Universal Robots PolyScope program: PSA_Tatiana.urp

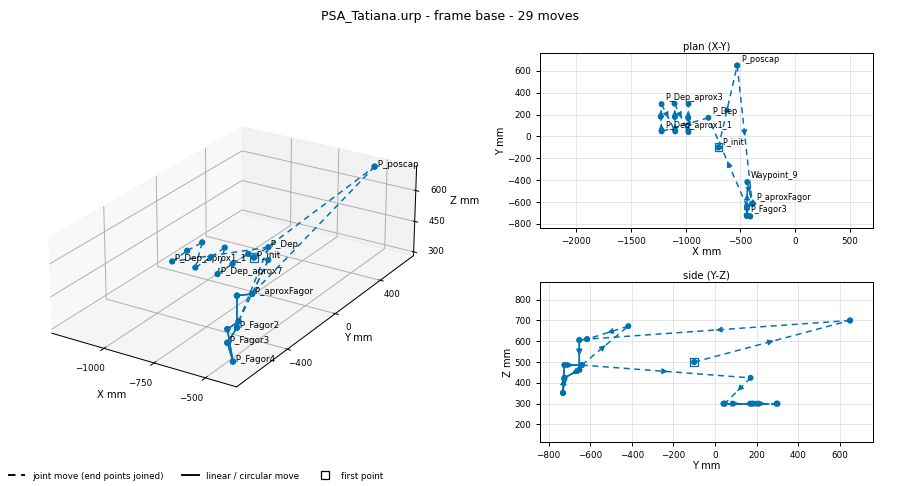
[picture p0: tool path of PSA_Tatiana.urp in frame base, 29 of 35 moves have a stored position in this frame; points joined in program order, loops and branches not executed]
Program PSA_Tatiana (installation=fbarreto directory=/programs/usbdisk createdIn=3.1.17195.0 lastSavedIn=3.15.3.106223 robotSerialNumber=2016302743)
Calibrated DH parameters: a=[0.000062, -0.599238, -0.569293, -0.000071, 0.00007, 0]; d=[0.127903, 43.80973, -52.244011, 8.598345, 0.115597, 0.092059]; alpha=[1.570295, -0.002885, -0.005578, 1.570526, -1.570968, 0]; deltaTheta=[0, -0.207803, 0.290321, -0.082351, -0.000076, 0.000026]
BeforeStart
  Set DigitalOutput pin=digital_out[1]; digitalValue=0
  RecolherPeca := False
  Set DigitalOutput pin=digital_out[2]; digitalValue=0
  RetirarPeca := False
  open := socket_open("192.168.114.51",5024)
  Loop While (checkContinuously=false) expression=open≟ False
    open := socket_open("192.168.114.51",5024)
  targetPos := p[0,0,0,0,0,0]
  '# Configuracao variaveis'
  var_from := p[0,0,0.05,0,0,0]
  var_from := p[0,0,-0.05,0,0,0]
  var_from := p[0.1,0,0,0,0,0]
  var_from := p[-0.1,0,0,0,0,0]
  P_dep_des := p[0,0,150/1000,0,0,0]
  P_dep_sub := p[0,0,-150/1000,0,0,0]
Robot Program (runOnlyOnce=false)
  '# Ligar Camara'
  Loop While (checkContinuously=false) expression=open≟ False
    open := socket_open("192.168.114.51",5024)
  Set DigitalOutput pin=digital_out[1]; digitalValue=1
  MoveJ speed 60 deg/s, acceleration 80 deg/s^2 (useActiveTCP=true)
    Waypoint P_init: TCP in base x=-700 y=-100 z=500 mm, rx=3.14 ry=0 rz=0 rad; joints [-5.413, -88.076, 103.177, -105.112, -90.206, -275.345] deg
    Loop While (checkContinuously=false) expression=RecolherPeca≟ False
      RecolherPeca := read_input_boolean_register(0)
    Waypoint P_poscap: TCP in base x=-528.533 y=649.105 z=699.93 mm, rx=2.2433 ry=-2.1967 rz=0 rad; joints [-62.276, -76.967, 70.287, -83.309, -90.248, -243.289] deg
  receiveFromServ := [0,0,0,0,0,0,0]
  SuppressedNode
    Wait Sleep waitTime=2
  receiveFromServ := socket_read_ascii_float(6)
  Loop While (checkContinuously=false) expression=receiveFromServ[0]≠6
    Wait Sleep waitTime=2
    sendToServer := "10@"
    Script: socket_send_string(sendToServer)
    receiveFromServ := socket_read_ascii_float(6)
  Folder GetCameraData Folder
    '# Here we should read the data from the camera'
    Ry := receiveFromServ[4]
    x_cam := receiveFromServ[2]
    y_cam := receiveFromServ[3]
    NewX := receiveFromServ[5]
    NewY := receiveFromServ[6]
  Folder Calculate Folder
    '# Convert mm to m and deg to rad'
    SuppressedNode
      Script file /programs/PSA_Tati_Pos.script
        | x=x_cam-x_cam*cos(Ry)
    target1 := p[x_cam/1000,y_cam/1000,0,0,0,0]
    target2 := p[0,0,0,0,0,Ry]
    target3 := p[NewX/1000,NewY/1000,0,0,0,0]
    target4 := p[0,0,285/1000,0,0,0]
  Folder MoveToCamPose
    MoveL speed 250 mm/s, acceleration 1200 mm/s^2 (useActiveTCP=false) tcp=TCP; feature=Joint_6_name
      Waypoint Waypoint (Variable): variable=target1
      Wait Sleep waitTime=0.5
      Waypoint Waypoint (Variable): variable=target2
      Wait Sleep waitTime=0.5
      Waypoint Waypoint (Variable): variable=target3
      Wait Sleep waitTime=0.5
      Waypoint Waypoint (Variable): variable=target4
      Set DigitalOutput pin=Ar; digitalValue=1
      Wait Sleep waitTime=2
      Waypoint P_poscap: motionParameters(blendRadius=0.05); TCP in base x=-528.533 y=649.105 z=699.93 mm, rx=2.2433 ry=-2.1967 rz=0 rad; joints [-62.276, -76.967, 70.287, -83.309, -90.248, -243.289] deg; pose in feature x=0 y=0 z=0 mm, rx=0 ry=0 rz=0 rad
  'Registo para PLC'
  Set DigitalOutput pin=digital_out[2]; digitalValue=1
  RecolherPeca := False
  Wait Sleep waitTime=0.1
  Set DigitalOutput pin=digital_out[2]; digitalValue=0
  'Movimentos para Fagor'
  MoveJ speed 60 deg/s, acceleration 80 deg/s^2 (useActiveTCP=true)
    SuppressedNode
      Waypoint P_init: TCP in base x=-700 y=-100 z=500 mm, rx=3.14 ry=0 rz=0 rad; joints [-5.413, -88.076, 103.177, -105.112, -90.206, -275.345] deg
    Waypoint P_aproxFagor: motionParameters(blendRadius=0.01); TCP in base x=-390.993 y=-615.089 z=610.275 mm, rx=2.1894 ry=-2.2258 rz=-0.0638 rad; joints [44.727, -87.76, 91.848, -95.173, -92.658, -134.226] deg
  MoveL speed 250 mm/s, acceleration 1200 mm/s^2 (useActiveTCP=true) feature=Base
    Waypoint P_Fagor1: motionParameters(blendRadius=0.05); TCP in base x=-439.397 y=-652.65 z=605.5 mm, rx=2.1896 ry=-2.2257 rz=-0.0637 rad; joints [44.175, -82.193, 86.245, -95.154, -92.662, -134.786] deg
    Waypoint P_Fagor2: motionParameters(blendRadius=0.05); TCP in base x=-439.462 y=-652.642 z=462.779 mm, rx=2.1897 ry=-2.2257 rz=-0.0637 rad; joints [44.183, -79.624, 97.856, -109.336, -92.647, -134.857] deg
    Waypoint P_Fagor3: motionParameters(blendRadius=0.029); TCP in base x=-440.419 y=-723.918 z=424.353 mm, rx=2.1893 ry=-2.2258 rz=-0.0638 rad; joints [47.686, -72.933, 93.423, -111.459, -92.725, -131.351] deg
    Waypoint P_Fagor4: TCP in base x=-409.469 y=-731.178 z=351.347 mm, rx=2.1897 ry=-2.2256 rz=-0.0643 rad; joints [49.639, -70.944, 98.714, -118.649, -92.761, -129.448] deg
    Set DigitalOutput pin=Ar; digitalValue=0
    Waypoint P_Fagor5: TCP in base x=-440.242 y=-724.015 z=485.586 mm, rx=2.1897 ry=-2.2257 rz=-0.0637 rad; joints [47.695, -74.653, 89.238, -105.541, -92.728, -131.322] deg
    Waypoint P_Fagor6: TCP in base x=-439.303 y=-640.298 z=485.545 mm, rx=2.1898 ry=-2.2259 rz=-0.0638 rad; joints [43.522, -81.208, 97.348, -107.258, -92.636, -135.506] deg
  'Registo para PLC'
  Set DigitalOutput pin=digital_out[3]; digitalValue=1
  Wait Sleep waitTime=0.1
  Set DigitalOutput pin=digital_out[3]; digitalValue=0
  'Esperar Maquinacao'
  MoveJ speed 60 deg/s, acceleration 80 deg/s^2 (useActiveTCP=true)
    Waypoint Waypoint_9: TCP in base x=-436.536 y=-416.989 z=672.545 mm, rx=2.1898 ry=-2.2258 rz=-0.0637 rad; joints [28.076, -100.049, 97.106, -88.753, -92.228, -150.869] deg
  Loop While (checkContinuously=false) expression=RetirarPeca≟ False
    RetirarPeca := read_input_boolean_register(2)
  SuppressedNode
    Wait Sleep waitTime=5
  MoveJ speed 60 deg/s, acceleration 80 deg/s^2 (useActiveTCP=true)
    SuppressedNode
      Waypoint P_init: TCP in base x=-700 y=-100 z=500 mm, rx=3.14 ry=0 rz=0 rad; joints [-5.413, -88.076, 103.177, -105.112, -90.206, -275.345] deg
    Waypoint P_aproxFagor: TCP in base x=-390.993 y=-615.089 z=610.275 mm, rx=2.1894 ry=-2.2258 rz=-0.0638 rad; joints [44.727, -87.76, 91.848, -95.173, -92.658, -134.226] deg
  MoveL speed 250 mm/s, acceleration 1200 mm/s^2 (useActiveTCP=true) feature=Base
    Waypoint P_Fagor1_1: motionParameters(blendRadius=0.05); TCP in base x=-439.397 y=-652.65 z=605.5 mm, rx=2.1896 ry=-2.2257 rz=-0.0637 rad; joints [44.175, -82.193, 86.245, -95.154, -92.662, -134.786] deg
    Waypoint P_Fagor2_1: motionParameters(blendRadius=0.05); TCP in base x=-439.462 y=-652.642 z=462.779 mm, rx=2.1897 ry=-2.2257 rz=-0.0637 rad; joints [44.183, -79.624, 97.856, -109.336, -92.647, -134.857] deg
    Waypoint P_Fagor3_1: motionParameters(blendRadius=0.029); TCP in base x=-440.419 y=-723.918 z=424.353 mm, rx=2.1893 ry=-2.2258 rz=-0.0638 rad; joints [47.686, -72.933, 93.423, -111.459, -92.725, -131.351] deg
    Waypoint P_Fagor4_2: TCP in base x=-409.469 y=-731.178 z=351.347 mm, rx=2.1897 ry=-2.2256 rz=-0.0643 rad; joints [49.639, -70.944, 98.714, -118.649, -92.761, -129.448] deg
    Set DigitalOutput pin=Ar; digitalValue=1
    Wait Sleep waitTime=2
    Waypoint P_Fagor5_1: motionParameters(blendRadius=0.05); TCP in base x=-440.242 y=-724.015 z=485.586 mm, rx=2.1897 ry=-2.2257 rz=-0.0637 rad; joints [47.695, -74.653, 89.238, -105.541, -92.728, -131.322] deg
    Waypoint P_Fagor6_1: motionParameters(blendRadius=0.032); TCP in base x=-439.303 y=-640.298 z=485.545 mm, rx=2.1898 ry=-2.2259 rz=-0.0638 rad; joints [43.522, -81.208, 97.348, -107.258, -92.636, -135.506] deg
  'Registo para PLC'
  Set DigitalOutput pin=digital_out[4]; digitalValue=1
  RetirarPeca := False
  Wait Sleep waitTime=0.1
  Set DigitalOutput pin=digital_out[4]; digitalValue=0
  MoveJ speed 60 deg/s, acceleration 80 deg/s^2 (useActiveTCP=true)
    Waypoint P_Dep: motionParameters(blendRadius=0.05); TCP in base x=-791.867 y=171.019 z=423.991 mm, rx=3.1339 ry=0.0381 rz=-0.1775 rad; joints [-24.299, -76.675, 99.441, -118.608, -87.451, -295.546] deg
  Set IncrementVariable installationVariable=Count_Deposito
  If Count_Deposito≟1
    MoveJ speed 60 deg/s, acceleration 80 deg/s^2 (useActiveTCP=true)
      Waypoint P_Dep_aprox1_1: motionParameters(blendRadius=0.005); TCP in base x=-1220.239 y=46.601 z=300 mm, rx=-3.0793 ry=-0.0321 rz=0.1301 rad; joints [-9.776, -31.849, 39.058, -102.603, -92.93, -281.068] deg
  ElseIf Count_Deposito≟2
    MoveJ speed 60 deg/s, acceleration 80 deg/s^2 (useActiveTCP=true)
      Waypoint P_Dep_aprox2: motionParameters(blendRadius=0.005); TCP in base x=-1227.991 y=180.872 z=300 mm, rx=-3.1238 ry=-0.0362 rz=0.1539 rad; joints [-16.089, -28.804, 33.23, -100.075, -89.6, -287.349] deg
  ElseIf Count_Deposito≟3
    MoveJ speed 60 deg/s, acceleration 80 deg/s^2 (useActiveTCP=true)
      Waypoint P_Dep_aprox3: motionParameters(blendRadius=0.005); TCP in base x=-1220.838 y=295.712 z=300 mm, rx=-3.1236 ry=-0.0361 rz=0.1539 rad; joints [-21.266, -26.027, 27.789, -97.317, -89.114, -292.49] deg
  ElseIf Count_Deposito≟4
    MoveJ speed 60 deg/s, acceleration 80 deg/s^2 (useActiveTCP=true)
      Waypoint P_Dep_apox4: motionParameters(blendRadius=0.005); TCP in base x=-1096.004 y=46.085 z=300 mm, rx=-3.1237 ry=-0.0363 rz=0.154 rad; joints [-11.116, -46.391, 66.072, -115.388, -90.028, -282.446] deg
  ElseIf Count_Deposito≟5
    MoveJ speed 60 deg/s, acceleration 80 deg/s^2 (useActiveTCP=true)
      Waypoint P_Dep_aprox5: motionParameters(blendRadius=0.005); TCP in base x=-1098.452 y=178.624 z=300 mm, rx=3.1402 ry=-0.0002 rz=-0.0009 rad; joints [-17.799, -44.326, 61.117, -106.816, -90.326, -287.758] deg
  ElseIf Count_Deposito≟6
    MoveJ speed 60 deg/s, acceleration 80 deg/s^2 (useActiveTCP=true)
      Waypoint P_Dep_aprox6: motionParameters(blendRadius=0.005); TCP in base x=-1102.071 y=300.706 z=300 mm, rx=3.1402 ry=0.0001 rz=-0.001 rad; joints [-23.6, -41.162, 55.369, -104.228, -90.337, -293.561] deg
  ElseIf Count_Deposito≟7
    MoveJ speed 60 deg/s, acceleration 80 deg/s^2 (useActiveTCP=true)
      Waypoint P_Dep_aprox7: motionParameters(blendRadius=0.005); TCP in base x=-974.911 y=40.045 z=300 mm, rx=3.1401 ry=-0.0001 rz=-0.0009 rad; joints [-12.13, -57.078, 83.145, -116.1, -90.266, -282.12] deg
  ElseIf Count_Deposito≟8
    MoveJ speed 60 deg/s, acceleration 80 deg/s^2 (useActiveTCP=true)
      Waypoint P_Dep_aprox8: motionParameters(blendRadius=0.005); TCP in base x=-976.81 y=168.063 z=300 mm, rx=3.1402 ry=-0.0001 rz=-0.0011 rad; joints [-19.387, -55.743, 80.934, -115.22, -90.274, -289.376] deg
  ElseIf Count_Deposito≟9
    MoveJ speed 60 deg/s, acceleration 80 deg/s^2 (useActiveTCP=true)
      Waypoint P_Dep_aprox9: motionParameters(blendRadius=0.005); TCP in base x=-974.391 y=297.299 z=300 mm, rx=3.1402 ry=0.0001 rz=-0.0007 rad; joints [-26.33, -53.311, 76.84, -113.537, -90.291, -296.32] deg
    Count_Deposito := 0
  MoveL speed 250 mm/s, acceleration 1200 mm/s^2 (useActiveTCP=false) tcp=TCP; feature=Joint_6_name
    SuppressedNode
      Waypoint P_Dep1: TCP in base x=-1230.762 y=59.351 z=139.091 mm, rx=-3.0793 ry=-0.0322 rz=0.1301 rad; joints [-10.285, -25.404, 42.948, -112.963, -92.875, -281.646] deg
    Waypoint Waypoint (Variable): variable=P_dep_des
    Set DigitalOutput pin=Ar; digitalValue=0
    Wait Sleep waitTime=1
    Waypoint Waypoint (Variable): motionParameters(blendRadius=0.05); variable=P_dep_sub
  Set DigitalOutput pin=digital_out[5]; digitalValue=1
  Wait Sleep waitTime=0.1
  Set DigitalOutput pin=digital_out[5]; digitalValue=0
  MoveJ speed 60 deg/s, acceleration 80 deg/s^2 (useActiveTCP=true)
    Waypoint P_init: motionParameters(blendRadius=0.05); TCP in base x=-700 y=-100 z=500 mm, rx=3.14 ry=0 rz=0 rad; joints [-5.413, -88.076, 103.177, -105.112, -90.206, -275.345] deg
